INTERFACE I_Test

METHOD METH : BOOL
VAR_INPUT
END_VAR
END_METHOD

PROPERTY Name : String
GET
END_GET
END_PROPERTY

END_INTERFACE

(* stored: Version 1.1.0.1, ProductVersion 3.1.4024.12
   Itf I_Test: Id {7b14dc32-22c2-45b1-b8cf-53a2660d831e}
   Method METH: Id {1bb01736-e5ad-44f3-b967-38c3a2aa8d6e}
   Property Name: Id {a59f8df2-f783-416d-961e-de7f7cabf77d}
   Get Get: Id {625e534f-1f6e-4911-bae0-f327927d32dc} *)
